{attribute 'TcGenerated'}
{attribute 'no-analysis'}
{attribute 'linkalways'}
// This function has been automatically generated from the project information.
VAR_GLOBAL CONSTANT
	{attribute 'const_non_replaced'}
	stLibVersion_PlantControl_and_CMs : ST_LibVersion := (iMajor := 0, iMinor := 1, iBuild := 0, iRevision := 0, nFlags := 0, sVersion := '0.1.0.0');
END_VAR

(* stored: Version 1.1.0.1, ProductVersion 3.1.4024.13
   GVL Global_Version: Id {76c5664a-406f-467e-8614-15b652bd511a} *)
